PROGRAM LateBlanking_Short_Test
VAR
ShortTest_Start_TON :Tc2_Standard.TON;	
TON_CYShort :Tc2_Standard.TON;
ShortTest_0: ShortTest;
Shortdata_ton :Tc2_Standard.TON;
YS_Short_ton :Tc2_Standard.TON;
FC_ton :Tc2_Standard.TON;
I:INT;
NG_Tim:Tc2_Standard.TON;
OK_Tim:Tc2_Standard.TON;
END_VAR

(*//短路测试//////////////////开通短路测试要删掉
IF Permit_ShortTest OR Shield[1] THEN
	CellMemory[CellNo.Hotpress].ShortTest:=1;
	ShortTest_Finish:=TRUE;
	Permit_ShortTest:=FALSE;
END_IF*)
shortcese();
ShortTest_Start_TON(PT:=T#8S);
TON_CYShort(PT:=T#6S);
Shortdata_ton(PT:=T#200MS);
YS_Short_ton(PT:=T#3.5S);
FC_ton(PT:=T#70MS);



//IF P3_SystemRUN.iMode=1  THEN//OR P3_SystemRUN.iMode=3
CASE Step_Short OF
0:
	TON_CYShort.IN:=FALSE;
	ShortTest_Start_TON.IN:=FALSE;
	arrCyCtrl[P3CYNo.P3ShortTest].Cmd.bOFF:=TRUE;
	P3Senser.P3_ShortTest_Start:=FALSE;
	Shortdata_ton.IN:=FALSE;
	YS_Short_ton.IN:=FALSE;	
	FC_ton.IN:=FALSE;
	I:=0;
	IF arrCyCtrl[P3CYNo.P3ShortTest].Status.OFFState AND NOT arrCyCtrl[P3CYNo.P3ShortTest].Status.Error2   THEN	
		Step_Short:=5;
	END_IF
5:
	IF  NOT ShortTest_Finish AND Permit_ShortTest AND arrAxisCtrl[P3AxisNo.P3_M3_HotPressingLine].Cmd.arrbRealPoint[2]
		 AND arrAxisCtrl[P3AxisNo.P3_M3_HotPressingLine].Status.NoMoving THEN
		Step_Short:=10;
	END_IF
10:
	IF P3User2_Par.Shield[1] THEN
		Step_Short:=0;
		ShortTest_Finish:=TRUE;	
		CellMemory[CellNo.Hotpress].ShortTest:=1;
	ELSIF Permit_ShortTest AND NOT ShortTest_Finish AND NOT P3Senser.P3_ShortTest_Testing AND Pressing[2] THEN
		 Step_Short:=20;
	END_IF 

20:
	TON_CYShort.IN:=TRUE;
    arrCyCtrl[P3CYNo.P3ShortTest].Cmd.bON:=TRUE;	
	IF (arrCyCtrl[P3CYNo.P3ShortTest].Status.ONState AND NOT arrCyCtrl[P3CYNo.P3ShortTest].Status.Error1) OR TON_CYShort.Q THEN	
	Step_Short:=30;
	TON_CYShort.IN:=FALSE;
	END_IF
		
30:
TON_CYShort.IN:=FALSE;
ShortTest_Start_TON.IN:=TRUE;
P3Senser.P3_ShortTest_Start:=TRUE;
IF ShortTest_Start_TON.Q THEN
Step_Short:=40;
ShortTest_Start_TON.IN:=FALSE;
END_IF

40:
ShortTest_Start_TON.IN:=FALSE;
Shortdata_ton.IN:=FALSE;
OK_Tim(IN:=P3Senser.P3_ShortTest_Pass , PT:=T#0.5S , Q=> , ET=> );
NG_Tim(IN:=P3Senser.P3_ShortTest_UpperFall OR P3Senser.P3_ShortTest_LowerFall , PT:=T#0.5S , Q=> , ET=> );
IF NG_Tim.Q THEN
//IF P3Senser.P3_ShortTest_UpperFall OR P3Senser.P3_ShortTest_LowerFall THEN
	CellMemory[CellNo.Hotpress].ShortTest:=2;
	NG_Tim(IN:=FALSE );
	Step_Short:=50;
	SHORT_HOT.bStart:=TRUE;
ELSIF OK_Tim.Q THEN
//ELSIF P3Senser.P3_ShortTest_Pass THEN
	CellMemory[CellNo.Hotpress].ShortTest:=1;
	OK_Tim(IN:=FALSE );
	Step_Short:=50;
	SHORT_HOT.bStart:=TRUE;	
END_IF

50:
Shortdata_ton.IN:=TRUE;
IF Shortdata_ton.Q AND SHORT_HOT.bDone THEN
Step_Short:=60;	
Shortdata_ton.IN:=FALSE;
END_IF

60:
CellMemory[CellNo.Hotpress].Hipot_R:=(SHORT_HOT.Measure);
CellMemory[CellNo.Hotpress].Hipot_Time:=SHORT_HOT.TestTime;
CellMemory[CellNo.Hotpress].Hipot_V:=SHORT_HOT.Voltage;
Step_Short:=70;	

70:
FC_ton.IN:=FALSE;
SHORT_HOT.bDone:=FALSE;
YS_Short_ton.IN:=FALSE;
P3Senser.P3_ShortTest_Start:=FALSE;
arrCyCtrl[P3CYNo.P3ShortTest].Cmd.bOFF:=TRUE;
Step_Short:=73;	

73:
IF ((CellMemory[CellNo.Hotpress].Hipot_R=0 AND CellMemory[CellNo.Hotpress].ShortTest<>2) 
OR CellMemory[CellNo.Hotpress].Hipot_Time=0 OR CellMemory[CellNo.Hotpress].Hipot_V=0) AND I<=3 THEN
	Step_Short:=1000;

	ELSIF ((CellMemory[CellNo.Hotpress].Hipot_R=0 AND CellMemory[CellNo.Hotpress].ShortTest<>2) 
OR CellMemory[CellNo.Hotpress].Hipot_Time=0 OR CellMemory[CellNo.Hotpress].Hipot_V=0) AND I>3 THEN
	Step_Short:=75;
	I:=0;
	CellMemory[CellNo.Hotpress].Hipot_R:=0;
	CellMemory[CellNo.Hotpress].ShortTest:=2;
	ELSE
	Step_Short:=75;
END_IF

(*
75:
	ShortTest_Finish:=TRUE;
	Permit_ShortTest:=FALSE;
	Step_Short:=0;	*)
75:
	IF NOT P3User2_Par.Shield[6] OR CellMemory[CellNo.Hotpress].ShortTest=2 THEN
		ShortTest_Finish:=TRUE;
		Permit_ShortTest:=FALSE;
		Step_Short:=0;	
	ELSE
	   Step_Short:=80;		
	END_IF



80:
YS_Short_ton.IN:=TRUE;	
IF YS_Short_ton.Q THEN
	arrCyCtrl[P3CYNo.P3ShortTest].Cmd.bON:=TRUE;
	YS_Short_ton.IN:=FALSE;
	TON_CYShort.IN:=TRUE;
	Step_Short:=90;
END_IF

90:
	IF TON_CYShort.Q THEN
		ShortTest_Start_TON.IN:=TRUE;
		P3Senser.P3_ShortTest_Start:=TRUE;
		TON_CYShort.IN:=FALSE;
		Step_Short:=100;
	END_IF
	
100:
	IF ShortTest_Start_TON.Q THEN
		Step_Short:=110;
		SHORT_HOT.bStart:=TRUE;
		ShortTest_Start_TON.IN:=FALSE;
	END_IF

110:
  IF P3Senser.P3_ShortTest_Pass AND CellMemory[CellNo.Hotpress].ShortTest=1 THEN
	  CellMemory[CellNo.Hotpress].ShortTest:=1;
	  Step_Short:=120;
	  ELSIF P3Senser.P3_ShortTest_UpperFall OR P3Senser.P3_ShortTest_LowerFall THEN
	   CellMemory[CellNo.Hotpress].ShortTest:=2;
	    Step_Short:=120;
  END_IF

120:
Shortdata_ton.IN:=TRUE;
IF Shortdata_ton.Q AND SHORT_HOT.bDone THEN
Step_Short:=130;	
Shortdata_ton.IN:=FALSE;
END_IF

130:
CellMemory[CellNo.Hotpress].Hipot2_R:=SHORT_HOT.Measure;
Step_Short:=140;	

140:
SHORT_HOT.bDone:=FALSE;
YS_Short_ton.IN:=FALSE;
P3Senser.P3_ShortTest_Start:=FALSE;
arrCyCtrl[P3CYNo.P3ShortTest].Cmd.bOFF:=TRUE;
ShortTest_Finish:=TRUE;
Permit_ShortTest:=FALSE;
Step_Short:=0;	
	
1000:
SHORT_HOT.bStart:=TRUE;
FC_ton.IN:=TRUE;
Step_Short:=1010;

1010:
IF  SHORT_HOT.bDone AND FC_ton.Q THEN
Step_Short:=60;	
FC_ton.IN:=FALSE;
I:=I+1;
END_IF



	
	
END_CASE
//END_IF

ACTION shortcese:
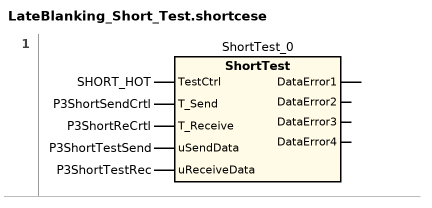
// NETWORK 1
ShortTest_0(
    TestCtrl := SHORT_HOT,
    T_Send := P3ShortSendCrtl,
    T_Receive := P3ShortReCrtl,
    uSendData := P3ShortTestSend,
    uReceiveData := P3ShortTestRec); // ShortTest
END_ACTION

END_PROGRAM

(* stored: Version 1.1.0.1, ProductVersion 3.1.4024.12
   POU LateBlanking_Short_Test: Id {e77788dc-a122-4d3b-adbc-e6cfaeb5cfe1}, SpecialFunc None
   Action shortcese: Id {155dd31c-7b45-4dec-a68e-b9094c678800} *)
